// TIA Portal V19 export
FUNCTION "CollectAlarms" : Void   // FC95, LAD
TITLE = Alarm Collector Unit
// Collects alarms from the respective level and categorises the alarms into the different alarm classes. Filling the alarm DB with specific alarm messages which are defined in the comment of the defined alarm. The definition of possible alarms within a equipment is handled here.
// stored: Namespace Unit2.EM4, SetENOAutomatically false
   VAR_INPUT
      resetAlarms : Bool;
      disableAlarms : Bool;
   END_VAR
   VAR_OUTPUT
      commandsToUnit : "LUC_typeStateCommands";   // Feedback to the unit
   END_VAR
   VAR_TEMP   // added for the SCL form of the ladder/FBD networks
      _w1 : Bool;
   END_VAR
BEGIN

REGION Network 1: Reset Alarms
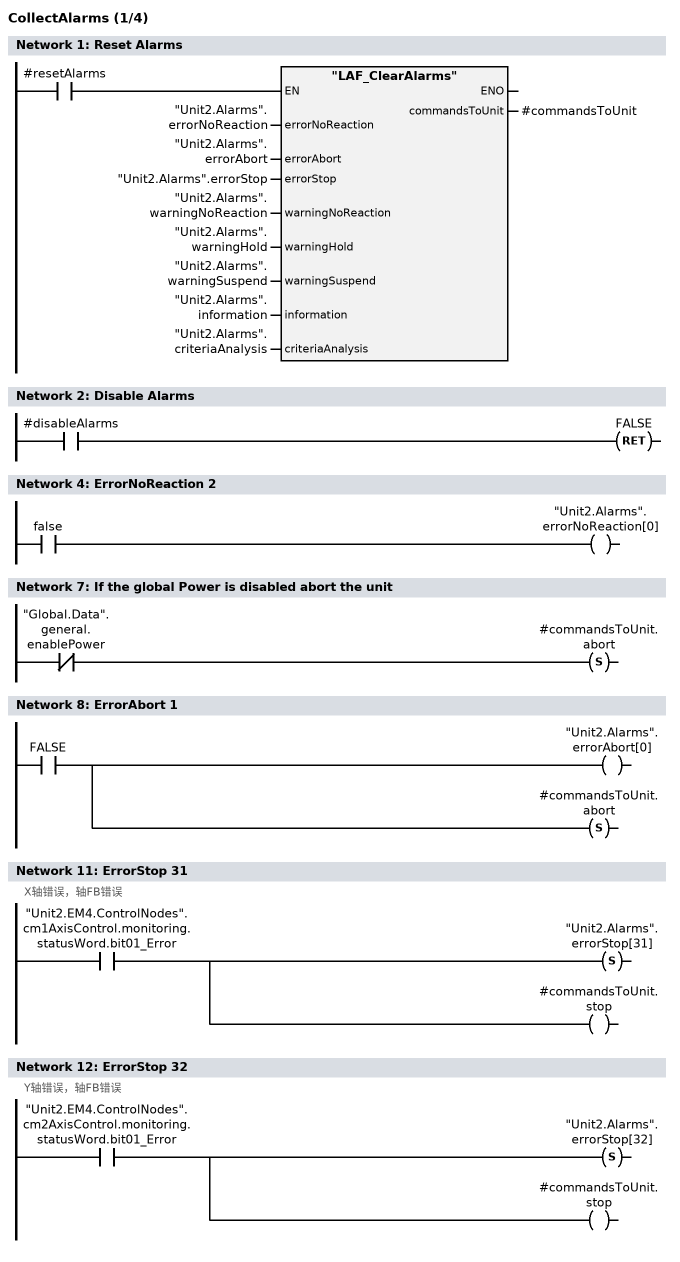
   RUNG wire#powerrail
      Contact( #resetAlarms )
      "LAF_ClearAlarms"(errorNoReaction := "Unit2.Alarms".errorNoReaction, errorAbort := "Unit2.Alarms".errorAbort, errorStop := "Unit2.Alarms".errorStop, warningNoReaction := "Unit2.Alarms".warningNoReaction, warningHold := "Unit2.Alarms".warningHold, warningSuspend := "Unit2.Alarms".warningSuspend, information := "Unit2.Alarms".information, criteriaAnalysis := "Unit2.Alarms".criteriaAnalysis, commandsToUnit => #commandsToUnit)
   END_RUNG
   // the same network as SCL:
   IF #resetAlarms THEN
       "LAF_ClearAlarms"(errorNoReaction := "Unit2.Alarms".errorNoReaction,
                         errorAbort := "Unit2.Alarms".errorAbort,
                         errorStop := "Unit2.Alarms".errorStop,
                         warningNoReaction := "Unit2.Alarms".warningNoReaction,
                         warningHold := "Unit2.Alarms".warningHold,
                         warningSuspend := "Unit2.Alarms".warningSuspend,
                         information := "Unit2.Alarms".information,
                         criteriaAnalysis := "Unit2.Alarms".criteriaAnalysis,
                         commandsToUnit => #commandsToUnit);
   END_IF;
END_REGION

REGION Network 2: Disable Alarms
   RUNG wire#powerrail
      Contact( #disableAlarms )
      ReturnCoil( FALSE )
   END_RUNG
   // the same network as SCL:
   IF #disableAlarms THEN
       ENO := FALSE;
       RETURN;
   END_IF;
END_REGION

REGION Network 3: *************** Error No Reaction ************************
END_REGION

REGION Network 4: ErrorNoReaction 2
   RUNG wire#powerrail
      Contact( false )
      Coil( "Unit2.Alarms".errorNoReaction[0] )
   END_RUNG
   // the same network as SCL:
   "Unit2.Alarms".errorNoReaction[0] := false;
END_REGION

REGION Network 6: *************** Error and Abort **************************
END_REGION

REGION Network 7: If the global Power is disabled abort the unit
   RUNG wire#powerrail
      I_Contact( "Global.Data".general.enablePower )
      S_Coil( #commandsToUnit.abort )
   END_RUNG
   // the same network as SCL:
   IF NOT "Global.Data".general.enablePower THEN #commandsToUnit.abort := TRUE; END_IF;
END_REGION

REGION Network 8: ErrorAbort 1
   RUNG wire#powerrail
      Contact( FALSE )
      wire#w1
      Coil( "Unit2.Alarms".errorAbort[0] )
   END_RUNG
   RUNG wire#w1
      S_Coil( #commandsToUnit.abort )
   END_RUNG
   // the same network as SCL:
   "Unit2.Alarms".errorAbort[0] := FALSE;
   IF FALSE THEN #commandsToUnit.abort := TRUE; END_IF;
END_REGION

REGION Network 10: *************** Error and Stop ***************************
END_REGION

REGION Network 11: ErrorStop 31
   // X轴错误，轴FB错误
   RUNG wire#powerrail
      Contact( "Unit2.EM4.ControlNodes".cm1AxisControl.monitoring.statusWord.bit01_Error )
      wire#w1
      S_Coil( "Unit2.Alarms".errorStop[31] )
   END_RUNG
   RUNG wire#w1
      Coil( #commandsToUnit.stop )
   END_RUNG
   // the same network as SCL:
   IF "Unit2.EM4.ControlNodes".cm1AxisControl.monitoring.statusWord.bit01_Error THEN
       "Unit2.Alarms".errorStop[31] := TRUE;
   END_IF;
   #commandsToUnit.stop := "Unit2.EM4.ControlNodes".cm1AxisControl.monitoring.statusWord.bit01_Error;
END_REGION

REGION Network 12: ErrorStop 32
   // Y轴错误，轴FB错误
   RUNG wire#powerrail
      Contact( "Unit2.EM4.ControlNodes".cm2AxisControl.monitoring.statusWord.bit01_Error )
      wire#w1
      S_Coil( "Unit2.Alarms".errorStop[32] )
   END_RUNG
   RUNG wire#w1
      Coil( #commandsToUnit.stop )
   END_RUNG
   // the same network as SCL:
   IF "Unit2.EM4.ControlNodes".cm2AxisControl.monitoring.statusWord.bit01_Error THEN
       "Unit2.Alarms".errorStop[32] := TRUE;
   END_IF;
   #commandsToUnit.stop := "Unit2.EM4.ControlNodes".cm2AxisControl.monitoring.statusWord.bit01_Error;
END_REGION

REGION Network 13: ErrorStop 33
   // Z轴错误，轴FB错误
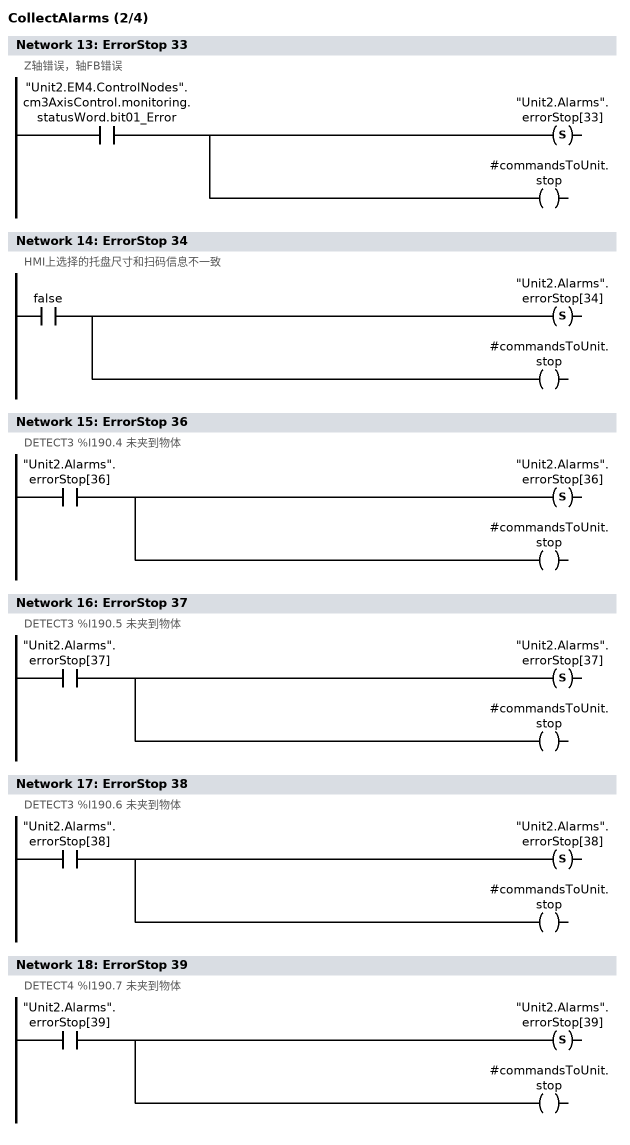
   RUNG wire#powerrail
      Contact( "Unit2.EM4.ControlNodes".cm3AxisControl.monitoring.statusWord.bit01_Error )
      wire#w1
      S_Coil( "Unit2.Alarms".errorStop[33] )
   END_RUNG
   RUNG wire#w1
      Coil( #commandsToUnit.stop )
   END_RUNG
   // the same network as SCL:
   IF "Unit2.EM4.ControlNodes".cm3AxisControl.monitoring.statusWord.bit01_Error THEN
       "Unit2.Alarms".errorStop[33] := TRUE;
   END_IF;
   #commandsToUnit.stop := "Unit2.EM4.ControlNodes".cm3AxisControl.monitoring.statusWord.bit01_Error;
END_REGION

REGION Network 14: ErrorStop 34
   // HMI上选择的托盘尺寸和扫码信息不一致
   RUNG wire#powerrail
      Contact( false )
      wire#w1
      S_Coil( "Unit2.Alarms".errorStop[34] )
   END_RUNG
   RUNG wire#w1
      Coil( #commandsToUnit.stop )
   END_RUNG
   // the same network as SCL:
   IF false THEN "Unit2.Alarms".errorStop[34] := TRUE; END_IF;
   #commandsToUnit.stop := false;
END_REGION

REGION Network 15: ErrorStop 36
   // DETECT3 %I190.4 未夹到物体
   RUNG wire#powerrail
      Contact( "Unit2.Alarms".errorStop[36] )
      wire#w1
      S_Coil( "Unit2.Alarms".errorStop[36] )
   END_RUNG
   RUNG wire#w1
      Coil( #commandsToUnit.stop )
   END_RUNG
   // the same network as SCL:
   #_w1 := "Unit2.Alarms".errorStop[36];
   IF #_w1 THEN "Unit2.Alarms".errorStop[36] := TRUE; END_IF;
   #commandsToUnit.stop := #_w1;
END_REGION

REGION Network 16: ErrorStop 37
   // DETECT3 %I190.5 未夹到物体
   RUNG wire#powerrail
      Contact( "Unit2.Alarms".errorStop[37] )
      wire#w1
      S_Coil( "Unit2.Alarms".errorStop[37] )
   END_RUNG
   RUNG wire#w1
      Coil( #commandsToUnit.stop )
   END_RUNG
   // the same network as SCL:
   #_w1 := "Unit2.Alarms".errorStop[37];
   IF #_w1 THEN "Unit2.Alarms".errorStop[37] := TRUE; END_IF;
   #commandsToUnit.stop := #_w1;
END_REGION

REGION Network 17: ErrorStop 38
   // DETECT3 %I190.6 未夹到物体
   RUNG wire#powerrail
      Contact( "Unit2.Alarms".errorStop[38] )
      wire#w1
      S_Coil( "Unit2.Alarms".errorStop[38] )
   END_RUNG
   RUNG wire#w1
      Coil( #commandsToUnit.stop )
   END_RUNG
   // the same network as SCL:
   #_w1 := "Unit2.Alarms".errorStop[38];
   IF #_w1 THEN "Unit2.Alarms".errorStop[38] := TRUE; END_IF;
   #commandsToUnit.stop := #_w1;
END_REGION

REGION Network 18: ErrorStop 39
   // DETECT4 %I190.7 未夹到物体
   RUNG wire#powerrail
      Contact( "Unit2.Alarms".errorStop[39] )
      wire#w1
      S_Coil( "Unit2.Alarms".errorStop[39] )
   END_RUNG
   RUNG wire#w1
      Coil( #commandsToUnit.stop )
   END_RUNG
   // the same network as SCL:
   #_w1 := "Unit2.Alarms".errorStop[39];
   IF #_w1 THEN "Unit2.Alarms".errorStop[39] := TRUE; END_IF;
   #commandsToUnit.stop := #_w1;
END_REGION

REGION Network 19: ErrorStop 40
   // 条件不满足，无法恢复步骤
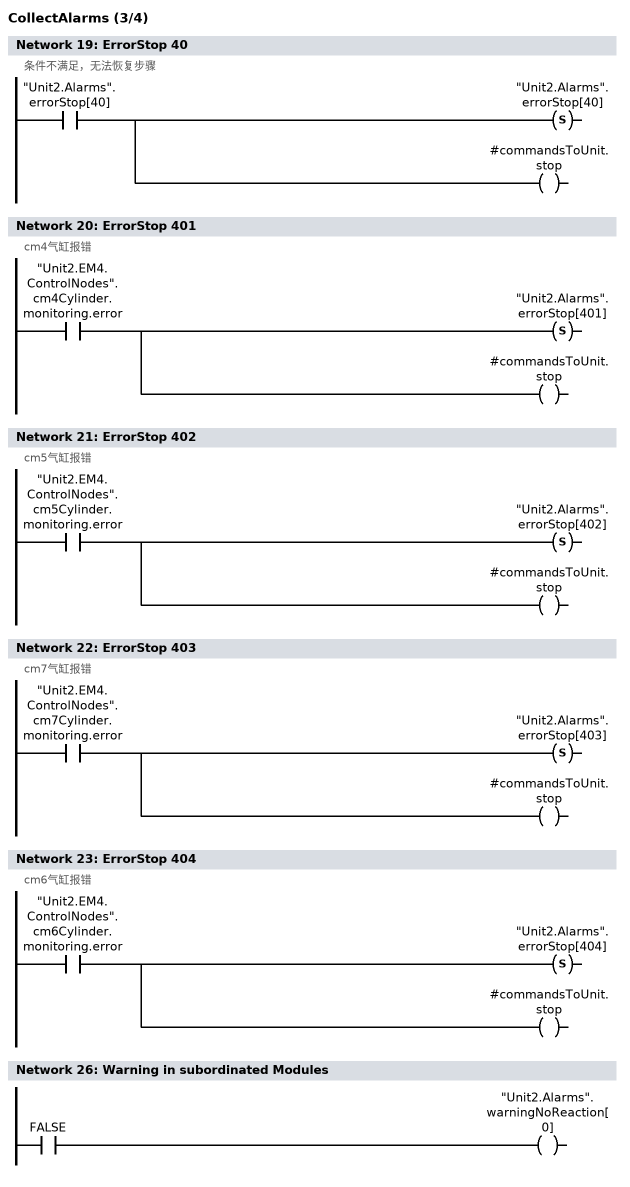
   RUNG wire#powerrail
      Contact( "Unit2.Alarms".errorStop[40] )
      wire#w1
      S_Coil( "Unit2.Alarms".errorStop[40] )
   END_RUNG
   RUNG wire#w1
      Coil( #commandsToUnit.stop )
   END_RUNG
   // the same network as SCL:
   #_w1 := "Unit2.Alarms".errorStop[40];
   IF #_w1 THEN "Unit2.Alarms".errorStop[40] := TRUE; END_IF;
   #commandsToUnit.stop := #_w1;
END_REGION

REGION Network 20: ErrorStop 401
   // cm4气缸报错
   RUNG wire#powerrail
      Contact( "Unit2.EM4.ControlNodes".cm4Cylinder.monitoring.error )
      wire#w1
      S_Coil( "Unit2.Alarms".errorStop[401] )
   END_RUNG
   RUNG wire#w1
      Coil( #commandsToUnit.stop )
   END_RUNG
   // the same network as SCL:
   IF "Unit2.EM4.ControlNodes".cm4Cylinder.monitoring.error THEN
       "Unit2.Alarms".errorStop[401] := TRUE;
   END_IF;
   #commandsToUnit.stop := "Unit2.EM4.ControlNodes".cm4Cylinder.monitoring.error;
END_REGION

REGION Network 21: ErrorStop 402
   // cm5气缸报错
   RUNG wire#powerrail
      Contact( "Unit2.EM4.ControlNodes".cm5Cylinder.monitoring.error )
      wire#w1
      S_Coil( "Unit2.Alarms".errorStop[402] )
   END_RUNG
   RUNG wire#w1
      Coil( #commandsToUnit.stop )
   END_RUNG
   // the same network as SCL:
   IF "Unit2.EM4.ControlNodes".cm5Cylinder.monitoring.error THEN
       "Unit2.Alarms".errorStop[402] := TRUE;
   END_IF;
   #commandsToUnit.stop := "Unit2.EM4.ControlNodes".cm5Cylinder.monitoring.error;
END_REGION

REGION Network 22: ErrorStop 403
   // cm7气缸报错
   RUNG wire#powerrail
      Contact( "Unit2.EM4.ControlNodes".cm7Cylinder.monitoring.error )
      wire#w1
      S_Coil( "Unit2.Alarms".errorStop[403] )
   END_RUNG
   RUNG wire#w1
      Coil( #commandsToUnit.stop )
   END_RUNG
   // the same network as SCL:
   IF "Unit2.EM4.ControlNodes".cm7Cylinder.monitoring.error THEN
       "Unit2.Alarms".errorStop[403] := TRUE;
   END_IF;
   #commandsToUnit.stop := "Unit2.EM4.ControlNodes".cm7Cylinder.monitoring.error;
END_REGION

REGION Network 23: ErrorStop 404
   // cm6气缸报错
   RUNG wire#powerrail
      Contact( "Unit2.EM4.ControlNodes".cm6Cylinder.monitoring.error )
      wire#w1
      S_Coil( "Unit2.Alarms".errorStop[404] )
   END_RUNG
   RUNG wire#w1
      Coil( #commandsToUnit.stop )
   END_RUNG
   // the same network as SCL:
   IF "Unit2.EM4.ControlNodes".cm6Cylinder.monitoring.error THEN
       "Unit2.Alarms".errorStop[404] := TRUE;
   END_IF;
   #commandsToUnit.stop := "Unit2.EM4.ControlNodes".cm6Cylinder.monitoring.error;
END_REGION

REGION Network 25: *************** Warning No Reaction **********************
END_REGION

REGION Network 26: Warning in subordinated Modules
   RUNG wire#powerrail
      Contact( FALSE )
      Coil( "Unit2.Alarms".warningNoReaction[0] )
   END_RUNG
   // the same network as SCL:
   "Unit2.Alarms".warningNoReaction[0] := FALSE;
END_REGION

REGION Network 27: WarningNoReaction 2
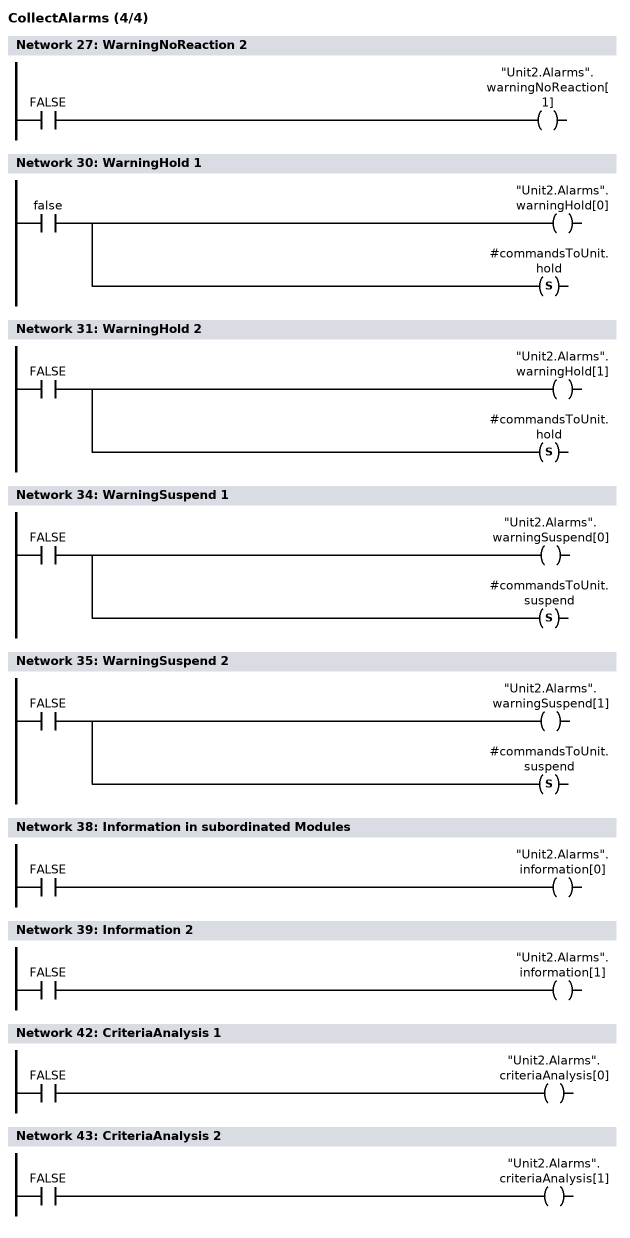
   RUNG wire#powerrail
      Contact( FALSE )
      Coil( "Unit2.Alarms".warningNoReaction[1] )
   END_RUNG
   // the same network as SCL:
   "Unit2.Alarms".warningNoReaction[1] := FALSE;
END_REGION

REGION Network 29: *************** Warning Hold **************************
END_REGION

REGION Network 30: WarningHold 1
   RUNG wire#powerrail
      Contact( false )
      wire#w1
      Coil( "Unit2.Alarms".warningHold[0] )
   END_RUNG
   RUNG wire#w1
      S_Coil( #commandsToUnit.hold )
   END_RUNG
   // the same network as SCL:
   "Unit2.Alarms".warningHold[0] := false;
   IF false THEN #commandsToUnit.hold := TRUE; END_IF;
END_REGION

REGION Network 31: WarningHold 2
   RUNG wire#powerrail
      Contact( FALSE )
      wire#w1
      Coil( "Unit2.Alarms".warningHold[1] )
   END_RUNG
   RUNG wire#w1
      S_Coil( #commandsToUnit.hold )
   END_RUNG
   // the same network as SCL:
   "Unit2.Alarms".warningHold[1] := FALSE;
   IF FALSE THEN #commandsToUnit.hold := TRUE; END_IF;
END_REGION

REGION Network 33: *************** Warning Suspend ***********************
END_REGION

REGION Network 34: WarningSuspend 1
   RUNG wire#powerrail
      Contact( FALSE )
      wire#w1
      Coil( "Unit2.Alarms".warningSuspend[0] )
   END_RUNG
   RUNG wire#w1
      S_Coil( #commandsToUnit.suspend )
   END_RUNG
   // the same network as SCL:
   "Unit2.Alarms".warningSuspend[0] := FALSE;
   IF FALSE THEN #commandsToUnit.suspend := TRUE; END_IF;
END_REGION

REGION Network 35: WarningSuspend 2
   RUNG wire#powerrail
      Contact( FALSE )
      wire#w1
      Coil( "Unit2.Alarms".warningSuspend[1] )
   END_RUNG
   RUNG wire#w1
      S_Coil( #commandsToUnit.suspend )
   END_RUNG
   // the same network as SCL:
   "Unit2.Alarms".warningSuspend[1] := FALSE;
   IF FALSE THEN #commandsToUnit.suspend := TRUE; END_IF;
END_REGION

REGION Network 37: *************** Information *****************************
END_REGION

REGION Network 38: Information in subordinated Modules
   RUNG wire#powerrail
      Contact( FALSE )
      Coil( "Unit2.Alarms".information[0] )
   END_RUNG
   // the same network as SCL:
   "Unit2.Alarms".information[0] := FALSE;
END_REGION

REGION Network 39: Information 2
   RUNG wire#powerrail
      Contact( FALSE )
      Coil( "Unit2.Alarms".information[1] )
   END_RUNG
   // the same network as SCL:
   "Unit2.Alarms".information[1] := FALSE;
END_REGION

REGION Network 41: *************** CriteriaAnalysis **************************
END_REGION

REGION Network 42: CriteriaAnalysis 1
   RUNG wire#powerrail
      Contact( FALSE )
      Coil( "Unit2.Alarms".criteriaAnalysis[0] )
   END_RUNG
   // the same network as SCL:
   "Unit2.Alarms".criteriaAnalysis[0] := FALSE;
END_REGION

REGION Network 43: CriteriaAnalysis 2
   RUNG wire#powerrail
      Contact( FALSE )
      Coil( "Unit2.Alarms".criteriaAnalysis[1] )
   END_RUNG
   // the same network as SCL:
   "Unit2.Alarms".criteriaAnalysis[1] := FALSE;
END_REGION
END_FUNCTION
